TYPE ST_SkillControl_2 :
STRUCT
    Start       : BOOL := FALSE;
    Cancel      : BOOL := FALSE;
    Reset       : BOOL := FALSE;

    RequestId   : UDINT := 0;
    Timeout     : REAL := 10.0;
END_STRUCT
END_TYPE

(* stored: Version 1.1.0.1, ProductVersion 3.1.4026.18
   DUT ST_SkillControl_2: Id {1f1fe46f-8422-49dc-a769-9a65bed25b07} *)
